// TIA Portal project "P1-01-Sorting-by-height" (V17)
// Sorting by height PLC Project using TIA Portal and Factory IO

(* hardware
DEVICE "S7-300/ET200M station_1"  S7-300 station
   slot 0: "Rail_0"  Rail  6ES7 390-1***0-0AA0
   slot 2: "PLC_1"  CPU 313C-2 DP  6ES7 313-6CG04-0AB0  V3.3
      slot 0: "MPI interface_1"  MPI
      slot 1: "DP interface_1"  DP
      slot 2: "DI 16/DO 16_1"  DI16/DO16
      slot 4: "Count_1"  Counter
*)

// ===== PLC "PLC_1"  CPU 313C-2 DP =====

VAR_GLOBAL   // PLC tag table "Default tag table"
   "High sensor" AT %I0.0 : Bool;
   "low sensor" AT %I0.1 : Bool;
   "pallet sensor" AT %I0.2 : Bool;
   "loaded sensor" AT %I0.3 : Bool;
   "at left entry" AT %I0.4 : Bool;
   "at right exit" AT %I0.7 : Bool;
   "start" AT %I1.0 : Bool;
   "reset" AT %I1.1 : Bool;
   "stop" AT %I1.2 : Bool;
   "emergency stop" AT %I1.3 : Bool;
   "auto" AT %I1.4 : Bool;
   "at right entry" AT %I0.6 : Bool;
   "at left exit" AT %I0.5 : Bool;
   "converyor entry" AT %Q0.0 : Bool;
   "load" AT %Q0.1 : Bool;
   "unload" AT %Q0.2 : Bool;
   "transfer left" AT %Q0.3 : Bool;
   "transfer right" AT %Q0.4 : Bool;
   "converyor left" AT %Q0.5 : Bool;
   "conveyor right" AT %Q0.6 : Bool;
   "start light" AT %Q0.7 : Bool;
   "reset light" AT %Q1.0 : Bool;
   "stop light" AT %Q1.1 : Bool;
   "a1" AT %M0.0 : Bool;
   "a2" AT %M0.1 : Bool;
   "Counter" AT %QW30 : Int;
END_VAR

ORGANIZATION_BLOCK "Main"   // OB1, LAD
TITLE = "Main Program Sweep (Cycle)"
{ S7_Optimized_Access := 'FALSE' }
VERSION : 0.1
   VAR_TEMP
      OB1_EV_CLASS : Byte;   // Bits 0-3 = 1 (Coming event), Bits 4-7 = 1 (Event class 1)
      OB1_SCAN_1 : Byte;   // 1 (Cold restart scan 1 of OB 1), 3 (Scan 2-n of OB 1)
      OB1_PRIORITY : Byte;   // Priority of OB Execution
      OB1_OB_NUMBR : Byte;   // 1 (Organization block 1, OB1)
      OB1_RESERVED_1 : Byte;   // Reserved for system
      OB1_RESERVED_2 : Byte;   // Reserved for system
      OB1_PREV_CYCLE : Int;   // Cycle time of previous OB1 scan (milliseconds)
      OB1_MIN_CYCLE : Int;   // Minimum cycle time of OB1 (milliseconds)
      OB1_MAX_CYCLE : Int;   // Maximum cycle time of OB1 (milliseconds)
      OB1_DATE_TIME : Date_And_Time;   // Date and time OB1 started
   END_VAR
   VAR_TEMP   // added for the SCL form of the ladder/FBD networks
      _w1 : Bool;
      _w2 : Bool;
   END_VAR
BEGIN

REGION Network 1
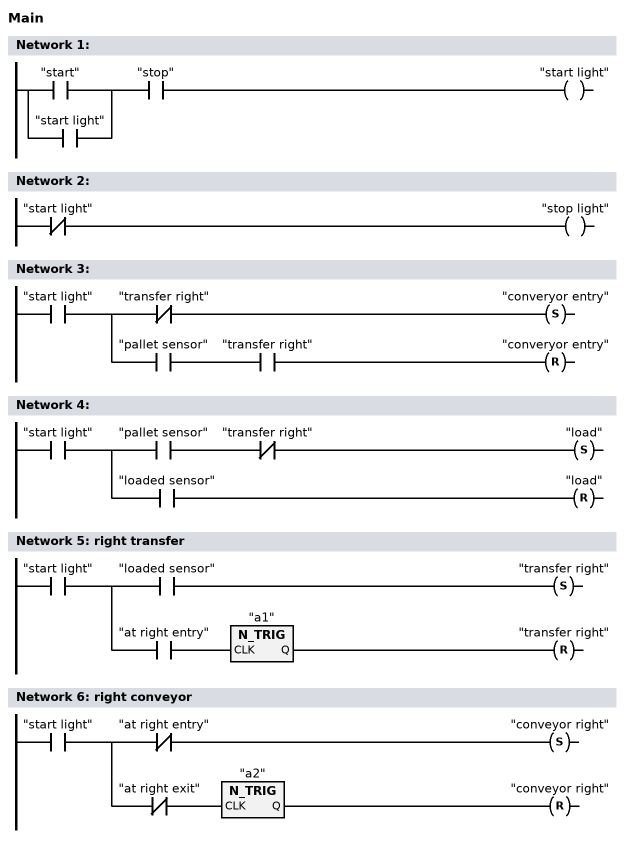
   RUNG wire#powerrail
      Contact( "start" )
      wire#w1
      Contact( "stop" )
      Coil( "start light" )
   END_RUNG
   RUNG wire#powerrail
      Contact( "start light" )
   END_RUNG wire#w1
   // the same network as SCL:
   "start light" := ("start" OR "start light") AND "stop";
END_REGION

REGION Network 2
   RUNG wire#powerrail
      I_Contact( "start light" )
      Coil( "stop light" )
   END_RUNG
   // the same network as SCL:
   "stop light" := NOT "start light";
END_REGION

REGION Network 3
   RUNG wire#powerrail
      Contact( "start light" )
      wire#w1
      I_Contact( "transfer right" )
      S_Coil( "converyor entry" )
   END_RUNG
   RUNG wire#w1
      Contact( "pallet sensor" )
      Contact( "transfer right" )
      R_Coil( "converyor entry" )
   END_RUNG
   // the same network as SCL:
   IF "start light" AND NOT "transfer right" THEN "converyor entry" := TRUE; END_IF;
   IF "start light" AND "pallet sensor" AND "transfer right" THEN "converyor entry" := FALSE; END_IF;
END_REGION

REGION Network 4
   RUNG wire#powerrail
      Contact( "start light" )
      wire#w1
      Contact( "pallet sensor" )
      I_Contact( "transfer right" )
      S_Coil( "load" )
   END_RUNG
   RUNG wire#w1
      Contact( "loaded sensor" )
      R_Coil( "load" )
   END_RUNG
   // the same network as SCL:
   IF "start light" AND "pallet sensor" AND NOT "transfer right" THEN "load" := TRUE; END_IF;
   IF "start light" AND "loaded sensor" THEN "load" := FALSE; END_IF;
END_REGION

REGION Network 5: right transfer
   RUNG wire#powerrail
      Contact( "start light" )
      wire#w1
      Contact( "loaded sensor" )
      S_Coil( "transfer right" )
   END_RUNG
   RUNG wire#w1
      Contact( "at right entry" )
      N_Trig( "a1" )
      R_Coil( "transfer right" )
   END_RUNG
   // the same network as SCL:
   IF "start light" AND "loaded sensor" THEN "transfer right" := TRUE; END_IF;
   #_w1 := "start light" AND "at right entry";
   #_w2 := NOT #_w1 AND "a1";   // falling edge
   "a1" := #_w1;
   IF #_w2 THEN "transfer right" := FALSE; END_IF;
END_REGION

REGION Network 6: right conveyor
   RUNG wire#powerrail
      Contact( "start light" )
      wire#w1
      I_Contact( "at right entry" )
      S_Coil( "conveyor right" )
   END_RUNG
   RUNG wire#w1
      I_Contact( "at right exit" )
      N_Trig( "a2" )
      R_Coil( "conveyor right" )
   END_RUNG
   // the same network as SCL:
   IF "start light" AND NOT "at right entry" THEN "conveyor right" := TRUE; END_IF;
   #_w1 := "start light" AND NOT "at right exit";
   #_w2 := NOT #_w1 AND "a2";   // falling edge
   "a2" := #_w1;
   IF #_w2 THEN "conveyor right" := FALSE; END_IF;
END_REGION
END_ORGANIZATION_BLOCK